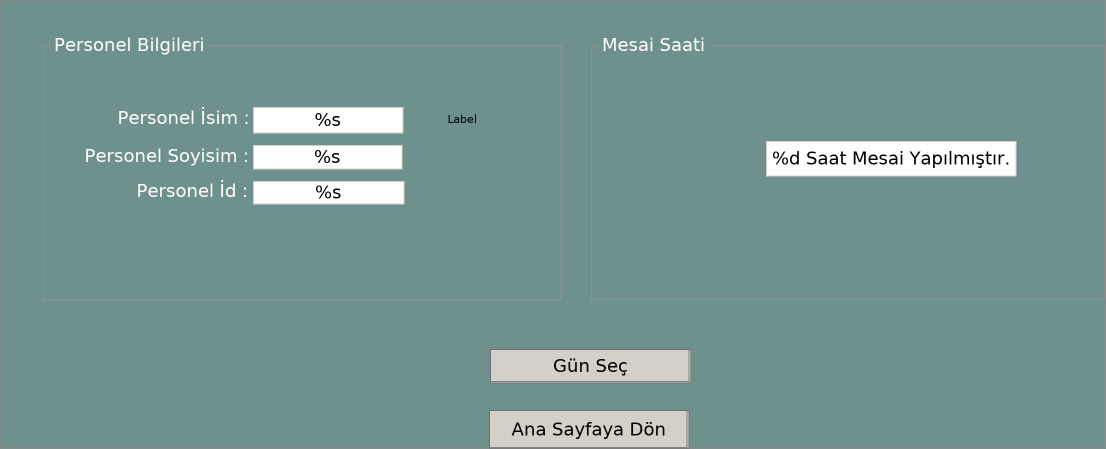
VISUALIZATION Hesap_Sayfa  // 1106x449
    GroupBox (43,37 518x263), "Personel Bilgileri"
        Label (69,66 143x30), "Personel İsim :"
        Label (44,104 160x30), "Personel Soyisim :"
        Label (78,139 143x30), "Personel İd :"
        Textfield (210,70 150x26), "%s", text variable: GVL_personel_kayit.perisim
        Textfield (210,108 149x24), "%s", text variable: GVL_personel_kayit.perSoyisim
        Textfield (210,144 151x23), "%s", text variable: GVL_personel_kayit.perid
    GroupBox (591,37 515x262), "Mesai Saati"
        Textfield (175,104 250x35), "%d Saat Mesai Yapılmıştır.", text variable: GVL_mesai_saat.tum_mesai
    Label (462,119 1x1), "Label"
    Button (490,349 201x34), "Gün Seç"
        OnMouseClick: change screen: mesaigunleri_sayfa
    Button (489,410 200x39), "Ana Sayfaya Dön"
        OnMouseClick: change screen: Ana_Sayfa
END_VISUALIZATION

(* stored: Version 1.1.0.1, ProductVersion 3.1.4024.12
   Visu Hesap_Sayfa: Id {56e1acc7-db4a-4c10-a247-47270fa3fe1e} *)
